Fanuc KAREL source: kf00117.KL

PROGRAM KF00117
%STACKSIZE=65535
%PRIORITY=65535
%NOLOCKGROUP
VAR
I : INTEGER
J : INTEGER
X : REAL
Y : REAL
B : BOOLEAN
C : BOOLEAN
TXT : STRING[80]
TXT2 : STRING[80]
AI : ARRAY[4] OF INTEGER
BI : ARRAY[4] OF INTEGER
P : XYZWPR
JP : JOINTPOS9
PF : POSITION
STATUS : INTEGER
-- UNRESOLVED DECLARATIONS (source type spelling not recovered)
-- V1 : TYPE_0x0013 (type_u16=0x0013)
-- V2 : TYPE_0x0013 (type_u16=0x0013)
ROUTINE PASSARR(P1 : ARRAY[*] OF INTEGER) FROM KF00117
ROUTINE PASSARR
BEGIN
I=P1[1]
END PASSARR
BEGIN
PASSARR(AI)
END KF00117
